// Mitsubishi GX Works2 project: plcGroup16_almostfinal   PLC: FX3G

// global labels: Global1
VAR_GLOBAL
  StartDay AT X007 : BOOL;
  OatMealInventory AT D1100 : REAL;
END_VAR
VAR_GLOBAL CONSTANT
  MinimumOatMeal : REAL := 399;
END_VAR
VAR_GLOBAL
  ProtienInventory AT D1102 : REAL;
END_VAR
VAR_GLOBAL CONSTANT
  MinimumProtien : REAL := 319;
END_VAR
VAR_GLOBAL
  EnoghOatMeal AT M1 : BOOL;
  EnoghProtien AT M2 : BOOL;
END_VAR
VAR_GLOBAL CONSTANT
  MinimumHoney : REAL := 159;
END_VAR
VAR_GLOBAL
  HoneyInventory AT D1104 : REAL;
  EnoghHoney AT M3 : BOOL;
  oatMealIndication AT M1 : BOOL;
  proteinIndication AT M2 : BOOL;
  honeyIndication AT M3 : BOOL;
  finishedPack AT Y004 : BOOL;
  EmergencyShutDown AT X005 : BOOL;
  startProduction AT M4 : BOOL;
  ifStillWorkDay AT Y000 : BOOL;
  INITIALDAY AT M4 : BOOL;
  oatMealCONTAINER AT D1106 : REAL;
  proteinCONTAINER AT D1108 : REAL;
  honeyCONTAINER AT D1110 : REAL;
  DAYSTARTED AT M5 : BOOL;
  MixStage AT X003 : BOOL;
  snackIndicator AT D8280 : INT;
  snackRegister AT D1120 : REAL;
  StartMIX AT M0 : BOOL;
  timerForMix AT TC10 : BOOL;
END_VAR
VAR_GLOBAL CONSTANT
  timerValue : INT := 50;
END_VAR
VAR_GLOBAL
  outputtimer AT TS10 : BOOL;
  MIXing AT Y003 : BOOL;
END_VAR
VAR_GLOBAL CONSTANT
  proteinvalue : REAL := 5;
END_VAR
VAR_GLOBAL
  proteinChosen AT M6 : BOOL;
END_VAR
VAR_GLOBAL CONSTANT
  clasicvalue : REAL := 5;
END_VAR
VAR_GLOBAL
  clasicChosen AT M7 : BOOL;
  randType AT D8282 : INT;
END_VAR
VAR_GLOBAL CONSTANT
  divide : REAL := 400;
  sub_oat : REAL := 240;
  sub_protein : REAL := 320;
  sub_honey : REAL := 160;
  sub_oat_c : REAL := 400;
  sub_protein_c : REAL := 160;
  sub_honey_c : REAL := 120;
END_VAR
VAR_GLOBAL
  bakeStage AT X002 : BOOL;
  baketIME_P AT TC20 : BOOL;
  BAKETime AT TC22 : BOOL;
END_VAR
VAR_GLOBAL CONSTANT
  baking_p : INT := 50;
  baking_c : INT := 40;
END_VAR
VAR_GLOBAL
  checknum309308950 AT Y001 : BOOL;
  ProteinBakingTime AT M8 : BOOL;
  ClassicBakingTime AT M9 : BOOL;
  startBulb AT M10 : BOOL;
  timerForBake AT TC12 : BOOL;
END_VAR
VAR_GLOBAL CONSTANT
  timetotimer : INT := 10;
END_VAR
VAR_GLOBAL
  outputTimer12 AT TS12 : BOOL;
  bulb_1 AT Y001 : BOOL;
  timer2 AT TC14 : BOOL;
  outputTimer14 AT TS14 : BOOL;
  bulb_2 AT Y002 : BOOL;
  checkcheck AT M76 : BOOL;
  outputtimer20 AT TS20 : BOOL;
  outputtimer22 AT TS22 : BOOL;
  packing_stage AT X006 : BOOL;
  pack_one_snack AT X000 : BOOL;
  CCpack AT CC1 : BOOL;
END_VAR
VAR_GLOBAL CONSTANT
  counterSnack : INT := 8;
END_VAR
VAR_GLOBAL
  destination AT M11 : BOOL;
  destination2 AT M12 : BOOL;
  Cspack AT CS1 : BOOL;
END_VAR
VAR_GLOBAL CONSTANT
  add_one : INT := 1;
END_VAR
VAR_GLOBAL
  num_packages AT D1200 : REAL;
END_VAR
VAR_GLOBAL CONSTANT
  COn40 : INT := 40;
END_VAR
VAR_GLOBAL
  num_packeges_output AT D8100 : INT;
  analog_output AT D8282 : INT;
  Conditionbake AT M20 : BOOL;
  conditionpack AT M40 : BOOL;
END_VAR

// task Task_01 (event TRUE, interval 0, priority 31): POU_01

PROGRAM POU_01
(* structured ladder/FBD written out as ST: instructions are called as NAME(EN, inputs, outputs); _pN, _eN, _tN stand for wires *)
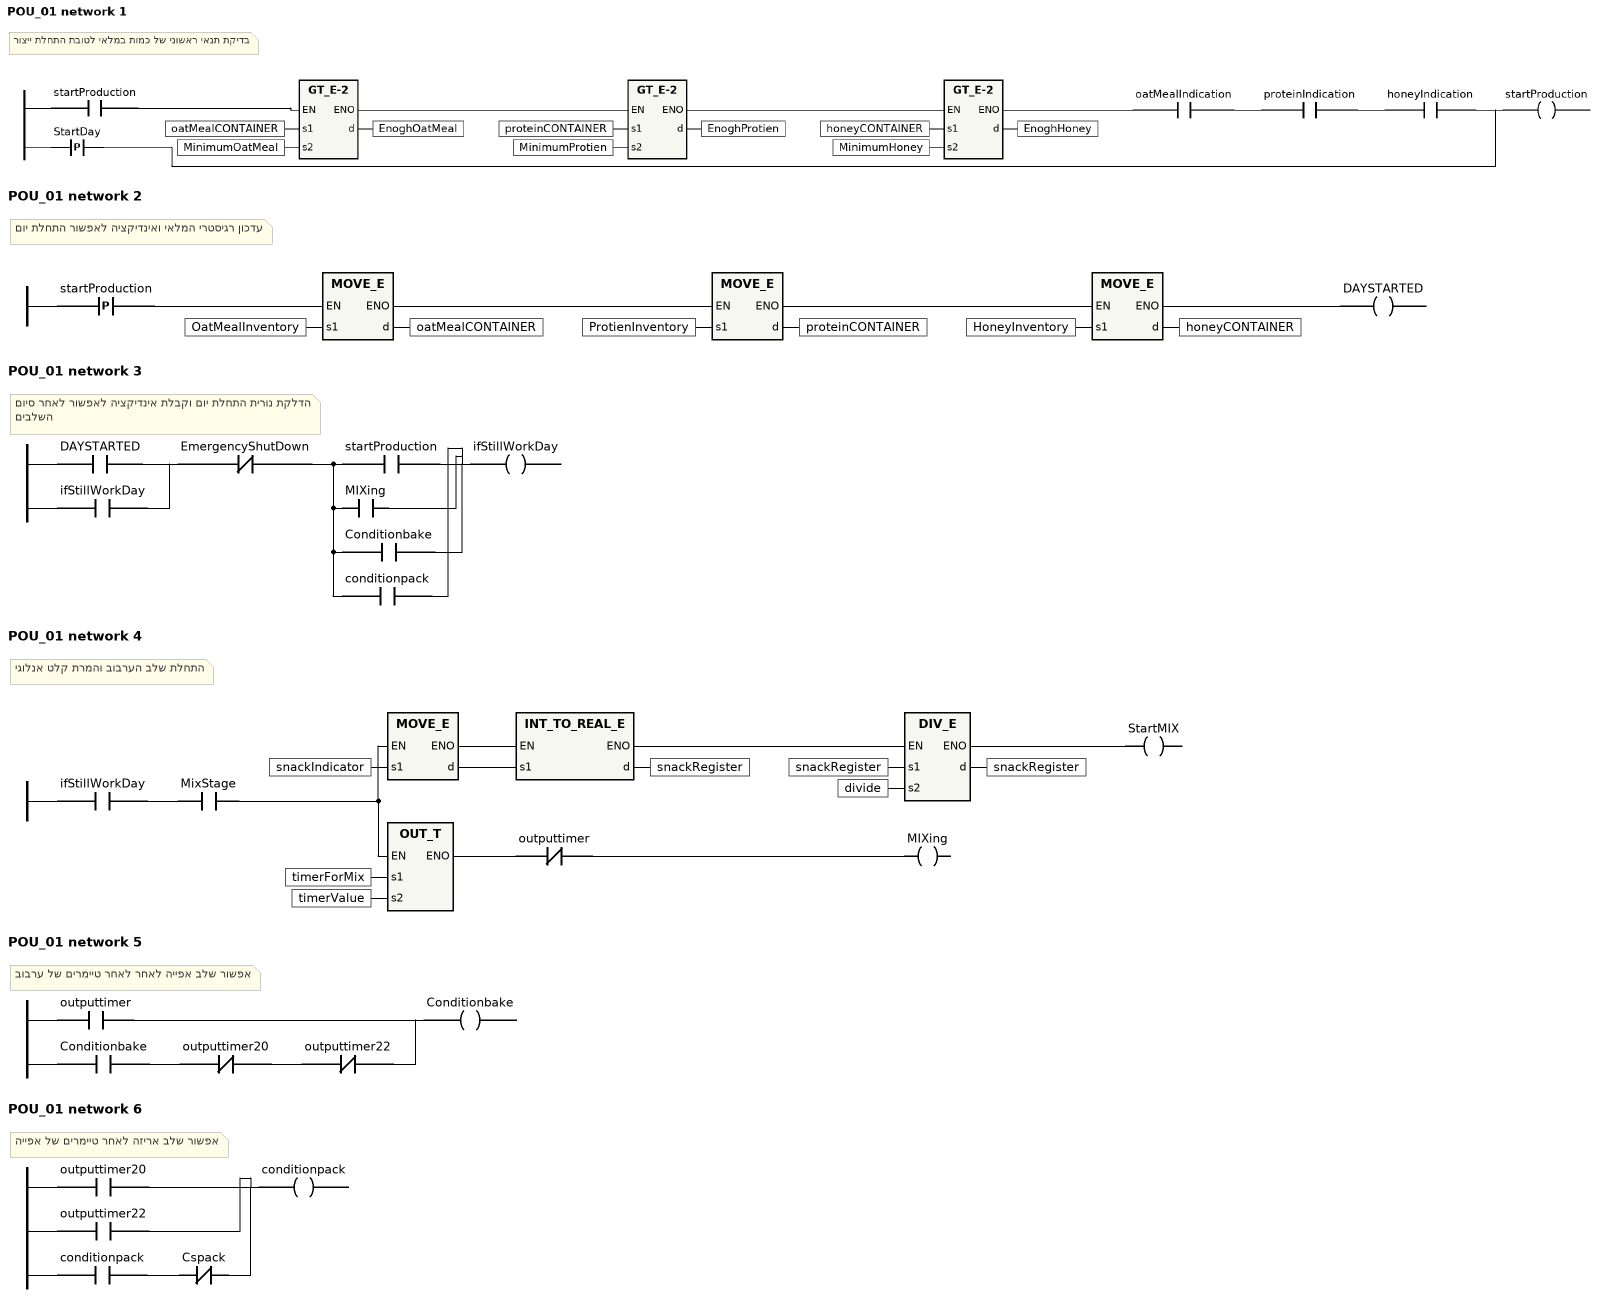
(* network 1 *)
(* בדיקת תנאי ראשוני של כמות במלאי לטובת התחלת ייצור *)
_e1 := GT_E(startProduction, oatMealCONTAINER, MinimumOatMeal, EnoghOatMeal);
_e2 := GT_E(_e1, proteinCONTAINER, MinimumProtien, EnoghProtien);
_e3 := GT_E(_e2, honeyCONTAINER, MinimumHoney, EnoghHoney);
startProduction := (_e3 AND oatMealIndication AND proteinIndication AND honeyIndication) OR LDP(TRUE, StartDay);
(* network 2 *)
(* עדכון רגיסטרי המלאי ואינדיקציה לאפשור התחלת יום *)
_e1 := MOVE_E(LDP(TRUE, startProduction), OatMealInventory, oatMealCONTAINER);
_e2 := MOVE_E(_e1, ProtienInventory, proteinCONTAINER);
_e3 := MOVE_E(_e2, HoneyInventory, honeyCONTAINER);
DAYSTARTED := _e3;
(* network 3 *)
(* הדלקת נורית התחלת יום וקבלת אינדיקציה לאפשור לאחר סיום השלבים *)
_p1 := (DAYSTARTED OR ifStillWorkDay) AND NOT EmergencyShutDown;
ifStillWorkDay := (_p1 AND startProduction) OR (_p1 AND MIXing) OR (_p1 AND Conditionbake) OR (_p1 AND conditionpack);
(* network 4 *)
(* התחלת שלב הערבוב והמרת קלט אנלוגי *)
_p1 := ifStillWorkDay AND MixStage;
_e3 := MOVE_E(_p1, snackIndicator, _t2);
_e4 := INT_TO_REAL_E(_e3, _t2, snackRegister);
_e5 := DIV_E(_e4, snackRegister, divide, snackRegister);
StartMIX := _e5;
_e6 := OUT_T(_p1, timerForMix, timerValue);
MIXing := _e6 AND NOT outputtimer;
(* network 5 *)
(* אפשור שלב אפייה לאחר לאחר טיימרים של ערבוב *)
Conditionbake := outputtimer OR (Conditionbake AND NOT outputtimer20 AND NOT outputtimer22);
(* network 6 *)
(* אפשור שלב אריזה לאחר טיימרים של אפייה *)
conditionpack := outputtimer20 OR outputtimer22 OR (conditionpack AND NOT Cspack);
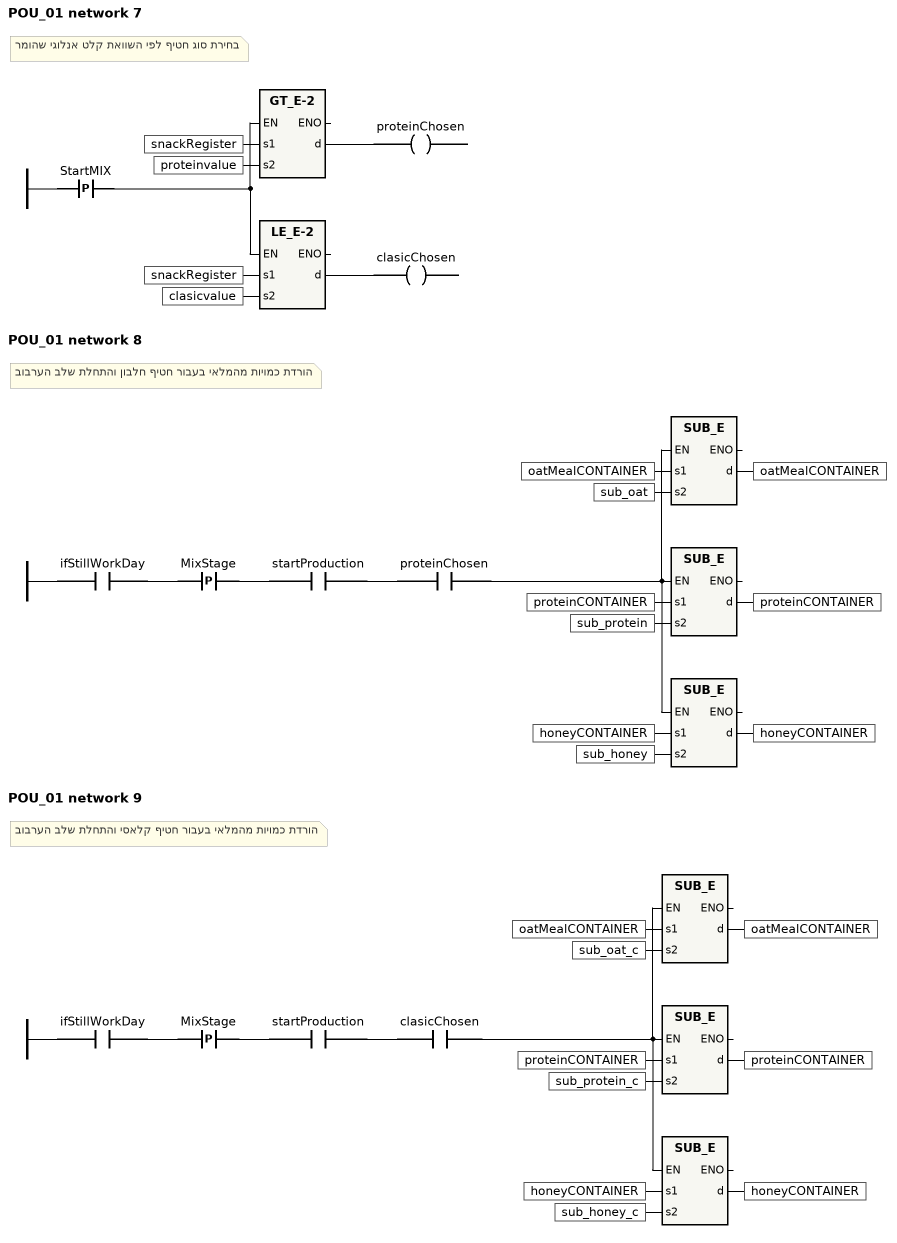
(* network 7 *)
(* בחירת סוג חטיף לפי השוואת קלט אנלוגי שהומר *)
_p1 := LDP(TRUE, StartMIX);
GT_E(_p1, snackRegister, proteinvalue, _t2);
proteinChosen := _t2;
LE_E(_p1, snackRegister, clasicvalue, _t3);
clasicChosen := _t3;
(* network 8 *)
(* הורדת כמויות מהמלאי בעבור חטיף חלבון והתחלת שלב הערבוב *)
_p1 := ifStillWorkDay AND LDP(TRUE, MixStage) AND startProduction AND proteinChosen;
SUB_E(_p1, oatMealCONTAINER, sub_oat, oatMealCONTAINER);
SUB_E(_p1, proteinCONTAINER, sub_protein, proteinCONTAINER);
SUB_E(_p1, honeyCONTAINER, sub_honey, honeyCONTAINER);
(* network 9 *)
(* הורדת כמויות מהמלאי בעבור חטיף קלאסי והתחלת שלב הערבוב *)
_p1 := ifStillWorkDay AND LDP(TRUE, MixStage) AND startProduction AND clasicChosen;
SUB_E(_p1, oatMealCONTAINER, sub_oat_c, oatMealCONTAINER);
SUB_E(_p1, proteinCONTAINER, sub_protein_c, proteinCONTAINER);
SUB_E(_p1, honeyCONTAINER, sub_honey_c, honeyCONTAINER);
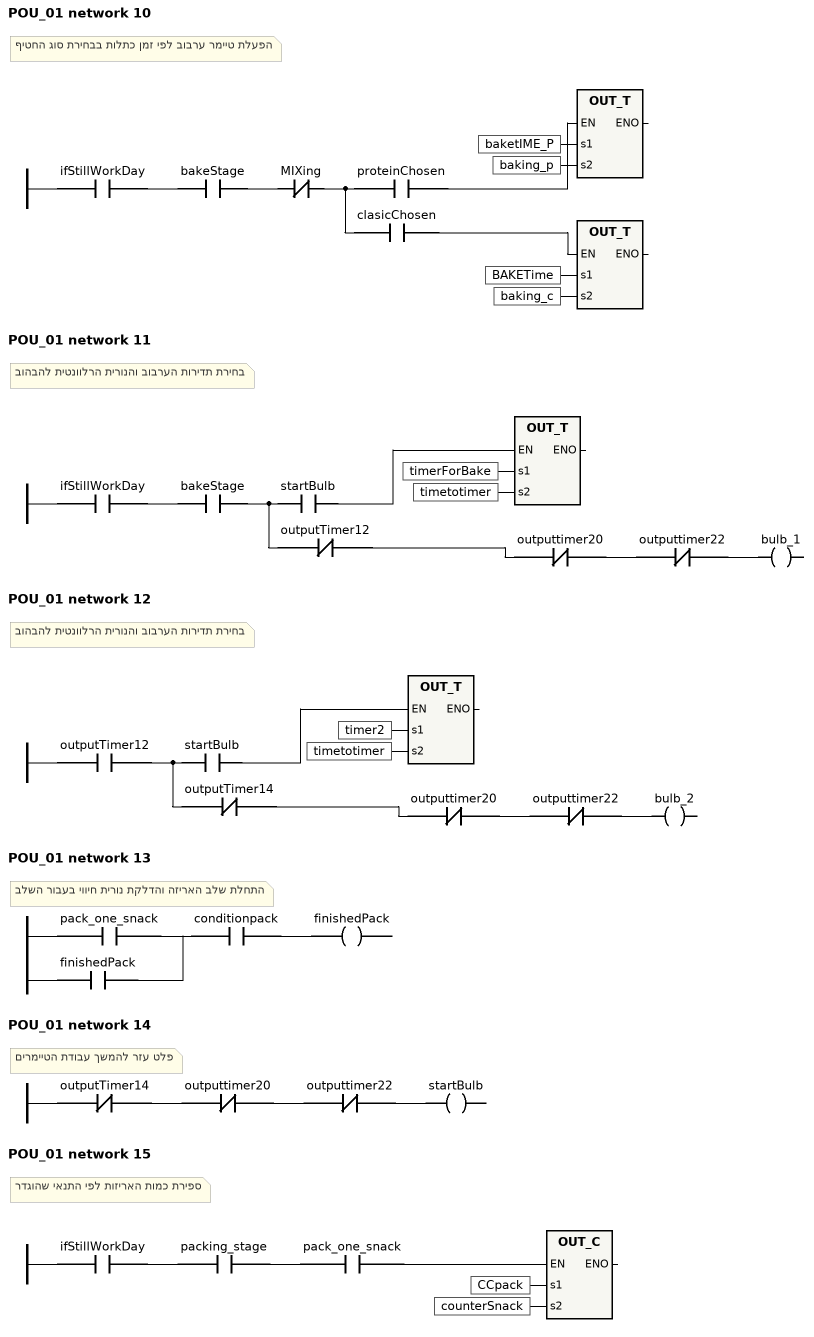
(* network 10 *)
(* הפעלת טיימר ערבוב לפי זמן כתלות בבחירת סוג החטיף *)
_p1 := ifStillWorkDay AND bakeStage AND NOT MIXing;
OUT_T(_p1 AND proteinChosen, baketIME_P, baking_p);
OUT_T(_p1 AND clasicChosen, BAKETime, baking_c);
(* network 11 *)
(* בחירת תדירות הערבוב והנורית הרלוונטית להבהוב *)
_p1 := ifStillWorkDay AND bakeStage;
OUT_T(_p1 AND startBulb, timerForBake, timetotimer);
bulb_1 := _p1 AND NOT outputTimer12 AND NOT outputtimer20 AND NOT outputtimer22;
(* network 12 *)
(* בחירת תדירות הערבוב והנורית הרלוונטית להבהוב *)
OUT_T(outputTimer12 AND startBulb, timer2, timetotimer);
bulb_2 := outputTimer12 AND NOT outputTimer14 AND NOT outputtimer20 AND NOT outputtimer22;
(* network 13 *)
(* התחלת שלב האריזה והדלקת נורית חיווי בעבור השלב *)
finishedPack := (pack_one_snack OR finishedPack) AND conditionpack;
(* network 14 *)
(* פלט עזר להמשך עבודת הטיימרים *)
startBulb := NOT outputTimer14 AND NOT outputtimer20 AND NOT outputtimer22;
(* network 15 *)
(* ספירת כמות האריזות לפי התנאי שהוגדר *)
OUT_C(ifStillWorkDay AND packing_stage AND pack_one_snack, CCpack, counterSnack);
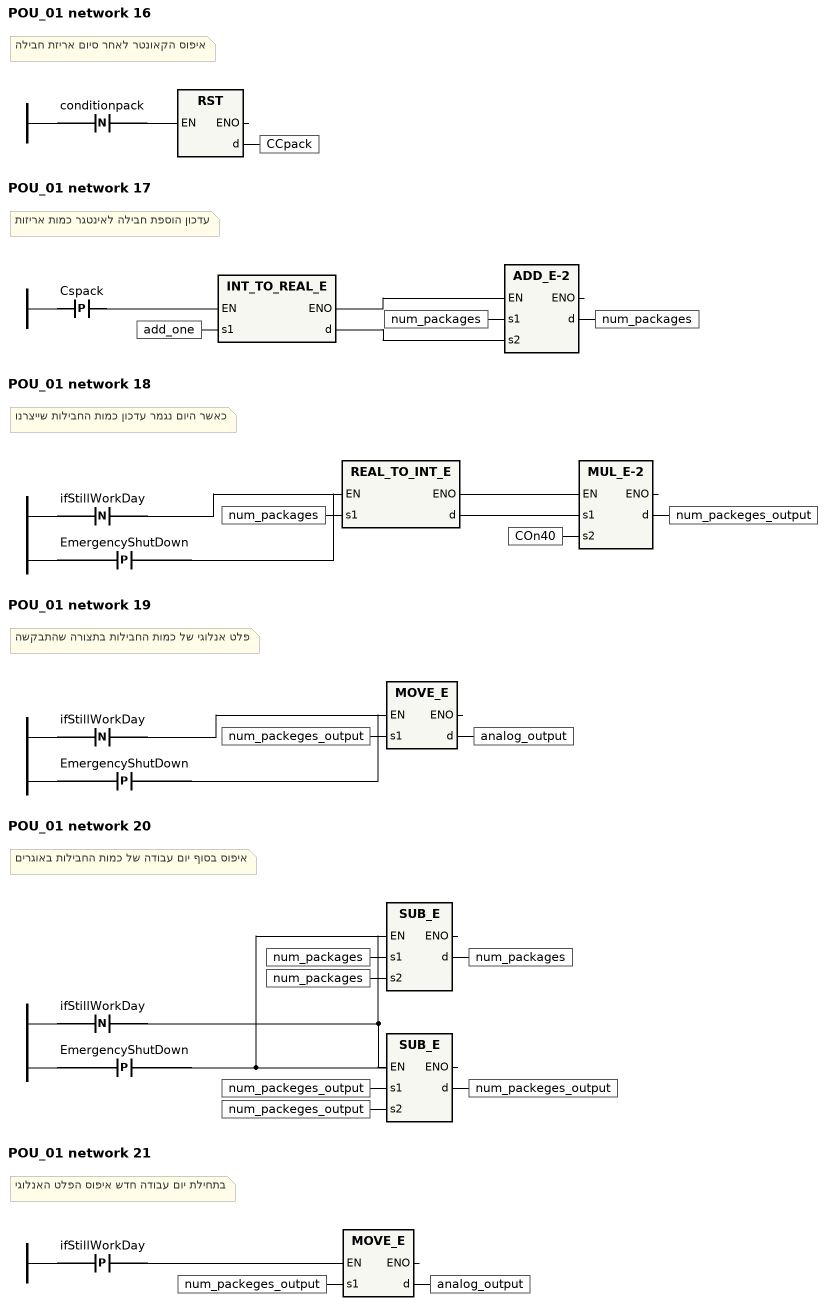
(* network 16 *)
(* איפוס הקאונטר לאחר סיום אריזת חבילה *)
RST(LDF(TRUE, conditionpack), CCpack);
(* network 17 *)
(* עדכון הוספת חבילה לאינטגר כמות אריזות *)
_e2 := INT_TO_REAL_E(LDP(TRUE, Cspack), add_one, _t1);
ADD_E(_e2, num_packages, _t1, num_packages);
(* network 18 *)
(* כאשר היום נגמר עדכון כמות החבילות שייצרנו *)
_e2 := REAL_TO_INT_E(LDF(TRUE, ifStillWorkDay) OR LDP(TRUE, EmergencyShutDown), num_packages, _t1);
MUL_E(_e2, _t1, COn40, num_packeges_output);
(* network 19 *)
(* פלט אנלוגי של כמות החבילות בתצורה שהתבקשה *)
MOVE_E(LDF(TRUE, ifStillWorkDay) OR LDP(TRUE, EmergencyShutDown), num_packeges_output, analog_output);
(* network 20 *)
(* איפוס בסוף יום עבודה של כמות החבילות באוגרים *)
_p1 := LDF(TRUE, ifStillWorkDay) OR LDP(TRUE, EmergencyShutDown);
SUB_E(_p1, num_packages, num_packages, num_packages);
SUB_E(_p1, num_packeges_output, num_packeges_output, num_packeges_output);
(* network 21 *)
(* בתחילת יום עבודה חדש איפוס הפלט האנלוגי *)
MOVE_E(LDP(TRUE, ifStillWorkDay), num_packeges_output, analog_output);
END_PROGRAM
